{attribute 'linkalways'} 
{attribute 'no_explicit_call' := 'This FB is a CLASS and must be accessed using methods or properties'}
{attribute 'enable_dynamic_creation'}
FUNCTION_BLOCK FINAL MODTURNS_LREAL EXTENDS Node
VAR
	value : _LREAL(0.0);
	arg : _LREAL(0.0);
	out : _DINT(0);
END_VAR

METHOD PUBLIC Clone : I_Node
VAR
	pNode : POINTER TO MODTURNS_LREAL;
END_VAR
pNode := __NEW(MODTURNS_LREAL);
Clone := pNode^;
END_METHOD

METHOD FB_init : BOOL
VAR_INPUT
	bInitRetains : BOOL; // if TRUE, the retain variables are initialized (warm start / cold start)
	bInCopyCode : BOOL;  // if TRUE, the instance afterwards gets moved into the copy code (online change)
END_VAR
AddInput('value',THIS^.value);
AddInput('arg',THIS^.arg);
AddOutput('out', THIS^.out);
END_METHOD

METHOD PROTECTED OnExecute
VAR
END_VAR
out.Value := MODTURNS(value.Value, arg.Value);
END_METHOD

END_FUNCTION_BLOCK

(* stored: Version 1.1.0.1, ProductVersion 3.1.4024.15
   POU MODTURNS_LREAL: Id {d27ba433-af6c-4e7e-8ba3-977cc4824588}, SpecialFunc None
   Folder Constructor: Id {aaad06ff-6a5f-462e-ada8-46aeb2e3d1e3}
   Method Clone: Id {21d325ca-4af2-4766-a76a-9be821a16739}
   Method FB_init: Id {9887e109-1572-4e89-8127-06ebed5c552f}
   Method OnExecute: Id {e1e92ed6-70f7-4c4d-866d-318080c7f476} *)
